{attribute 'qualified_only'}
VAR_GLOBAL	
	B1 AT %Q*: BOOL;	// Endschalter Offen
	B2 AT %Q*: BOOL;   // Endschalter Geschlossen
	B3 AT %Q*: BOOL;   // Lichtschranke
	S1 AT %Q*: BOOL;   // Taster "Halt"
	S2 AT %Q*: BOOL;   // Taster "Öffnen"
	S3 AT %Q*: BOOL;   // Taster "Schliessen"
END_VAR

(* stored: Version 1.1.0.1, ProductVersion 3.1.4024.5
   GVL DI: Id {c2d05302-d374-4f85-80dd-41006a3e3277} *)
